# EPICS autosave request: soft_iocs/galil_DMC/iocBoot/iocgalil_DMC_A01/slit_settings.req
file "2slit_soft_settings.req", P=$(P), SLIT=XenocsUS_V:
file "2slit_soft_settings.req", P=$(P), SLIT=XenocsUS_H:
